{attribute 'strict'}
TYPE E_ContactorError :
(
	CONTACTOR_ERROR_OK := 0,
	CONTACTOR_ERROR_MOVE_ACTIVE_TIMED_OUT := 20
);
END_TYPE

(* stored: Version 1.1.0.1, ProductVersion 3.1.4024.12
   DUT E_ContactorError: Id {233b670d-e1d4-4861-88b3-bef3f0e4a969} *)
